{attribute 'no_check'}
//Simple object for one hardware output with an additionl bit to forward the Out status to the AT  %Q* variable
FUNCTION_BLOCK Output 
VAR_INPUT
	Enable													:	BOOL := TRUE;	//FB will be processed as long as enable is TRUE 	
	Out														:	BOOL := FALSE;	//sets output
END_VAR         								
VAR_OUTPUT      								
	status													:	BYTE := 0;		//query Options (conditions see below)
	Q												AT  %Q* :	BOOL;			//hardware output
END_VAR         							
VAR             				
END_VAR

IF Out THEN
	switchOn();
ELSE
	SwitchOff();
END_IF

status.0 													:= NOT Q;
status.1 													:= Q;
status.5 													:= Enable;

METHOD PUBLIC switchOff : booL
VAR_INPUT
END_VAR
Q := Out											:= FALSE;
SwitchOff											:= TRUE;
END_METHOD

METHOD PUBLIC switchOn : booL
VAR_INPUT
END_VAR
Out														:= TRUE;
SwitchOn := Q 											:= Enable AND Out;
END_METHOD

END_FUNCTION_BLOCK

(* stored: Version 1.1.0.1, ProductVersion 3.1.4024.3
   POU Output: Id {bfc4f4e5-dbe0-41dd-9de3-68ac105cf38e}, SpecialFunc None
   Method switchOff: Id {7a803ce3-62fc-4d11-b256-e7afcdaa7d24}
   Method switchOn: Id {d845a3e4-f40a-4cb9-89a0-c12196b98144} *)
